// TIA Portal V20 export
FUNCTION_BLOCK "Fault"   // FB304, FBD
{ S7_Optimized_Access := 'TRUE' }
// stored: AutoNumber false, MemoryReserve 100, SetENOAutomatically false
   VAR
      Var : "TypeVar";
      T : Array[1..16] of IEC_TIMER;
      ErrSafetyModule { ExternalAccessible := 'False'; ExternalVisible := 'False'; ExternalWritable := 'False'} : Bool;
   END_VAR
BEGIN

REGION Network 1: fault acknowledge - pc
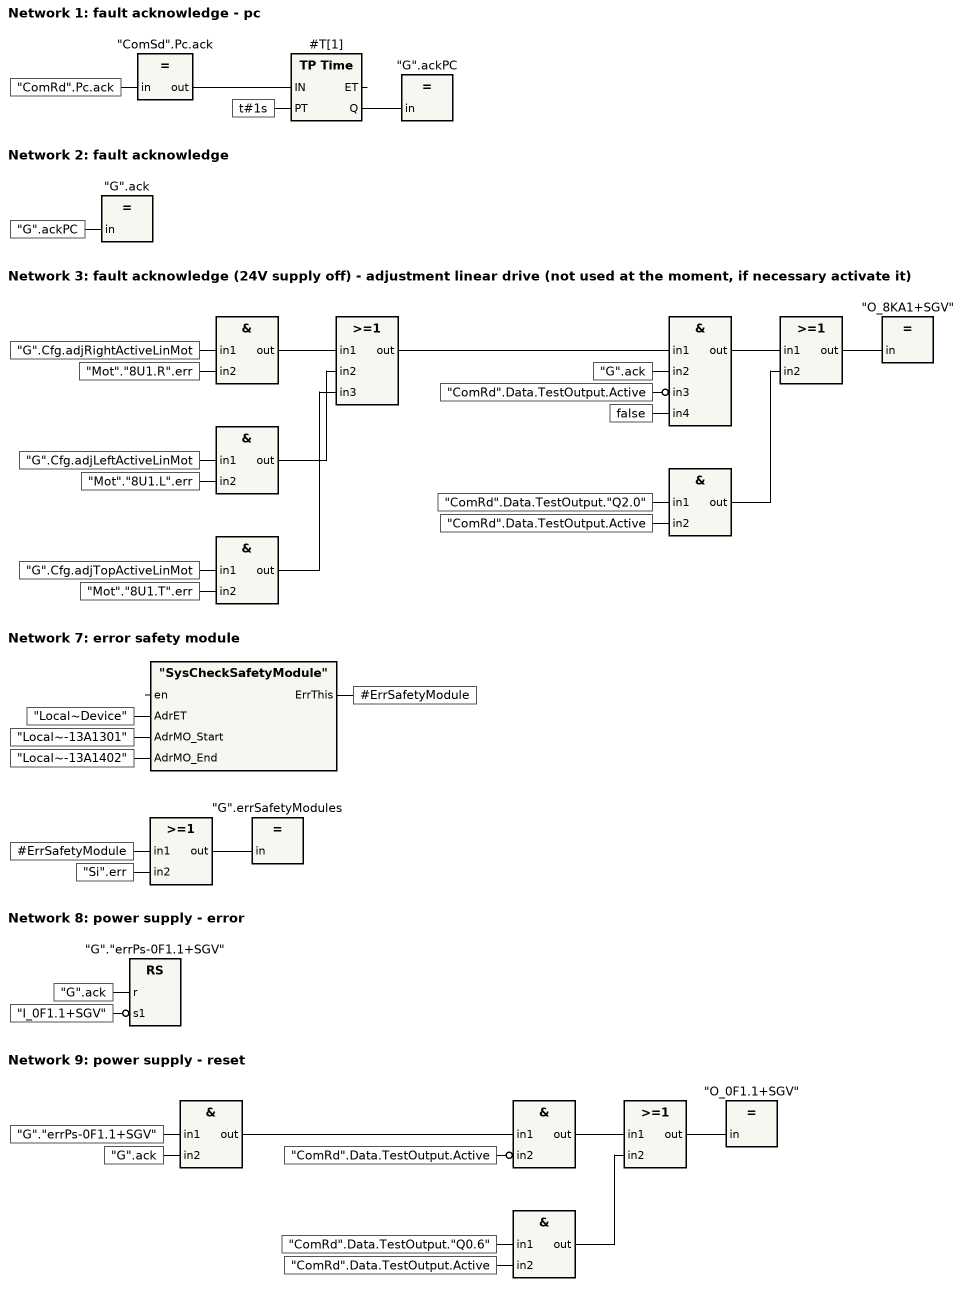
   "ComSd".Pc.ack := "ComRd".Pc.ack;
   #T[1].TP(IN := "ComRd".Pc.ack, PT := t#1s);
   "G".ackPC := #T[1].Q;
END_REGION

REGION Network 2: fault acknowledge
   "G".ack := "G".ackPC;
END_REGION

REGION Network 3: fault acknowledge (24V supply off) - adjustment linear drive (not used at the moment, if necessary activate it)
   "O_8KA1+SGV" := ((("G".Cfg.adjRightActiveLinMot AND "Mot"."8U1.R".err) OR ("G".Cfg.adjLeftActiveLinMot AND "Mot"."8U1.L".err) OR ("G".Cfg.adjTopActiveLinMot AND "Mot"."8U1.T".err)) AND "G".ack AND NOT "ComRd".Data.TestOutput.Active AND false) OR ("ComRd".Data.TestOutput."Q2.0" AND "ComRd".Data.TestOutput.Active);
END_REGION

NETWORK
TITLE = info general
      O     "false";

      =     "G".info;

NETWORK
TITLE = warning general
      O     "Si".settingModeActive;
      O     "Si".jogModeActive;
      O     "I_0SH1+SSTR";

      =     "G".war;

NETWORK
TITLE = fault general
// fault safety
      O     "G".errSafetyModules;
      O     "Si".aLaserErrFdb;
      O     "Si".aAdjustmentErrFdb1;
      O     "Si".aAdjustmentErrFdb2;
      O(;
      A     "Si".aXrayErrFdb;
      A     "G".Cfg.xrayActive;
      );

// fault communication / pc
      O     "G".errComPc;
      O     "G".errVersion;

// fault power supply
      O     "G"."errPs-0F1.1+SGV";
      O     "G"."errAc-0E1+SGV";
      O     "G"."errAc-0E2+SGX";
      O     "G"."errAc-0E1.1+SGV";

// fault profinet
      O     "G".errProfinet;

// fault sensor
      O     "Sen"."1BTR2+SGV".err;
      O     "Sen"."1BTR2+SGX".err;

// fault encoder
      O     "Enc"."1BCI1".err;
      O     "Enc"."1BCM1".err;
      O     "Enc"."1BCO1".err;

// fault motor
      O     "G".errAdjScanner;
      O     "G".errAdjTop;
      O     "G".errAdjLeft;
      O     "G".errAdjRight;

      O     "false";
      =     "G".err;

REGION Network 7: error safety module
   "SysCheckSafetyModule"(AdrET := "Local~Device",
                          AdrMO_Start := "Local~-13A1301",
                          AdrMO_End := "Local~-13A1402",
                          ErrThis => #ErrSafetyModule);
   "G".errSafetyModules := #ErrSafetyModule OR "Si".err;
END_REGION

REGION Network 8: power supply - error
   IF "G".ack THEN
       "G"."errPs-0F1.1+SGV" := FALSE;   // RS flip-flop
   END_IF;
   IF NOT "I_0F1.1+SGV" THEN "G"."errPs-0F1.1+SGV" := TRUE; END_IF;
END_REGION

REGION Network 9: power supply - reset
   "O_0F1.1+SGV" := ("G"."errPs-0F1.1+SGV" AND "G".ack AND NOT "ComRd".Data.TestOutput.Active) OR ("ComRd".Data.TestOutput."Q0.6" AND "ComRd".Data.TestOutput.Active);
END_REGION

REGION Network 10: fault profinet device
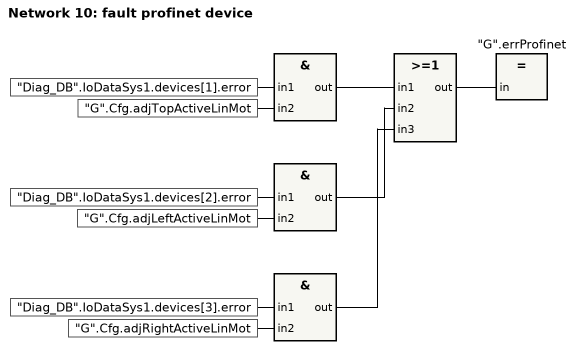
   "G".errProfinet := ("Diag_DB".IoDataSys1.devices[1].error AND "G".Cfg.adjTopActiveLinMot) OR ("Diag_DB".IoDataSys1.devices[2].error AND "G".Cfg.adjLeftActiveLinMot) OR ("Diag_DB".IoDataSys1.devices[3].error AND "G".Cfg.adjRightActiveLinMot);
END_REGION
END_FUNCTION_BLOCK
